// TwinCAT 3 PLC project Example
// ProgramVersion: 3.1.4023.0
// libraries:
//   Tc2_Standard, * (Beckhoff Automation GmbH)
//   Tc2_System, * (Beckhoff Automation GmbH)
//   Tc3_Module, * (Beckhoff Automation GmbH)
//   Twinson, * (Stefan Besler)
// project tree:
//   / PlcTask.TcTTO
//   POUs/ MAIN.TcPOU
// real-time tasks:
//   TASK PlcTask: cycle T#10ms, priority 20, ADS port 350

CONFIGURATION Example
    RESOURCE PLC ON TwinCAT3
        TASK PlcTask(INTERVAL := T#10ms, PRIORITY := 20);
        PROGRAM MAIN WITH PlcTask : MAIN;
    END_RESOURCE
END_CONFIGURATION

// ---- POUs/MAIN.TcPOU
PROGRAM MAIN
VAR
  json : Twinson.JsonDecoder;
  parse : BOOL := TRUE;
END_VAR

IF parse
THEN
  parse := FALSE;
  json.DecodeText('{ "integer1": 5, "string1": "la", "null1": null, "object1" : { "subint1":5, "substring1":"lala", "subfloat1":5.44 }, "string2": "asdf"  }');  
END_IF

END_PROGRAM
